PROGRAM MAIN
VAR
	count1 :INT;
	F1 :FBDelayCheck;
END_VAR


F1(in := count1, delaytime := T#0.2S);

END_PROGRAM

(* stored: Version 1.1.0.1, ProductVersion 3.1.4022.18
   POU MAIN: Id {331e9dbf-c59d-4b03-a4cc-cb4fe771a8ab}, SpecialFunc None *)
